Yaskawa INFORM job: TEST-DATA.JBI

/JOB
//NAME TEST-DATA
//POS
///NPOS 0,0,0,0,0,0
//INST
///DATE 2018/09/27 08:50
///ATTR SC,RW
///GROUP1 RB1
NOP
MACRO1 MJ#(1) ARGF1 ARGF10
PAUSE
MACRO1 MJ#(1) ARGF2 ARGF6
PAUSE
MACRO1 MJ#(1) ARGF3 ARGF9
PAUSE
MACRO1 MJ#(1) ARGF4 ARGF5
PAUSE
MACRO1 MJ#(1) ARGF5 ARGF7
PAUSE
MACRO1 MJ#(1) ARGF8 ARGF60
PAUSE
MACRO1 MJ#(1) ARGF9 ARGF61
PAUSE
MACRO1 MJ#(1) ARGF10 ARGF67
PAUSE
MACRO1 MJ#(2) ARGF100 ARGF68
PAUSE
MACRO1 MJ#(2) ARGF101 ARGF68
PAUSE
MACRO1 MJ#(2) ARGF102 ARGF68
PAUSE
MACRO1 MJ#(2) ARGF103 ARGF68
PAUSE
MACRO1 MJ#(2) ARGF20 ARGF70
PAUSE
MACRO1 MJ#(2) ARGF21 ARGF71
PAUSE
MACRO1 MJ#(2) ARGF22 ARGF70
PAUSE
MACRO1 MJ#(2) ARGF23 ARGF71
PAUSE
MACRO1 MJ#(2) ARGF24 ARGF35
PAUSE
MACRO1 MJ#(2) ARGF25 ARGF36
PAUSE
MACRO1 MJ#(2) ARGF26 ARGF35
PAUSE
MACRO1 MJ#(2) ARGF27 ARGF36
PAUSE
MACRO1 MJ#(2) ARGF28 ARGF54
PAUSE
MACRO1 MJ#(2) ARGF29 ARGF54
END
